FUNCTION TryConvert_TOD_TO_STRING : BOOL
VAR_INPUT
	in : TOD;
	out : REFERENCE TO STRING;
END_VAR

out := TOD_TO_STRING(in);
TryConvert_TOD_TO_STRING := TRUE;

END_FUNCTION

(* stored: Version 1.1.0.1, ProductVersion 3.1.4024.12
   POU TryConvert_TOD_TO_STRING: Id {e4c8f674-fc62-42ce-a744-f4e8758a83f9}, SpecialFunc None *)
